{attribute 'GeneratedUsingTerminal: KL3351-0003'}
{attribute addProperty BoxType "KL3351-0003"}
{attribute addProperty Id "StatusAT %I*USINT0Ud_RegInAT %I*INT0UrefAT %I*INT0CtrlAT %Q*USINT0RegOutAT %Q*INT0Ctrl1AT %Q*USINT0"}
{attribute addProperty CRC "85240058"}
{attribute addProperty Size "0"}
TYPE Channel_0514A8FA :
STRUCT
	{attribute addProperty Name "Status"}
	Status AT %I* : USINT;
	{attribute addProperty Name "Ud_RegIn"}
	Ud_RegIn AT %I* : INT;
	{attribute addProperty Name "Uref"}
	Uref AT %I* : INT;
	{attribute addProperty Name "Ctrl"}
	Ctrl AT %Q* : USINT;
	{attribute addProperty Name "RegOut"}
	RegOut AT %Q* : INT;
	{attribute addProperty Name "Ctrl1"}
	Ctrl1 AT %Q* : USINT;
END_STRUCT
END_TYPE

(* stored: Version 1.2.0.0, ProductVersion 3.1.4024.9
   DUT Channel_0514A8FA: Id {be55125a-07ea-4897-ada3-b6000120e418} *)
